Staubli VAL3: ROBERT_TP6.pjx

--- ROBERT_TP6.pjx ---
Parameters version=s7.9 stackSize=5000 millimeterUnit=true
Program file=Poche.pgx
Program file=start.pgx
Program file=stop.pgx
Data file=ROBERT_TP6.dtx

--- ROBERT_TP6.dtx ---
mdesc mRapide100On
mdesc mUsinage20Off = {vel=20, blend=off}
jointRx jStart = {j1=-13.1554864532824, j2=52.8057266959055, j3=128.56179776802, j4=166.840895901009, j5=91.3316286241402, j6=-180.311296989427}
tool tBroche = {x=169.400168374358, y=5.67105066906493E-05, z=47.7499999146672, ry=90, rz=90, fatherId=flange[0], ioLink=valve1}
num nDiametreFraise = 10
frame fPiece = {x=527.606812, y=-37.435701, z=-438.0625, rx=180, rz=-90, fatherId=world[0]}
pointRx pStartUsinage = {x=25, y=25, fatherId=fPiece[0]}
jointRx jChangeOutil = {j1=-4.70104777967739, j2=85.6578357974361, j3=60.0632848818122, j4=174.316678572801, j5=55.8523989241203, j6=-80.7639740285582}
trsf trAppro = {z=-22}
num nPasseRadiale
mdesc mUsinage5Off = {vel=5, blend=off}

--- start.pgx ---
program start()
begin
  resetMotion()
  movej(jStart, tBroche, mRapide100On)

  call Poche(pStartUsinage, nDiametreFraise, 7, 4, 100, 50, 20)

  movej(jChangeOutil, tBroche, mRapide100On)
  waitEndMove()
end

--- Poche.pgx ---
program Poche(pointRx x_pStartPoint, num x_nDiametreTool, num x_nPasseAxiale, num x_nPasseRadiale, num x_nDimX, num x_nDimY, num x_nDimZ)
  local num l_nIndex
  local pointRx l_pPoint[5]
  local num l_nIndex2
  local num l_nN
  local num l_nLongueurCote
  local num l_nIndex3
  local num l_nM
  local num l_nProfondeur
begin
  logMsg("Beginning...")

  l_nProfondeur = x_nDimZ

  l_nN = roundDown((x_nDimX-x_nDiametreTool-x_nPasseRadiale)/(2*x_nPasseRadiale)+1)
  l_nM = roundDown(l_nProfondeur/(x_nPasseAxiale))

  for l_nIndex3 = 1 to l_nM
    logMsg("New passe...")
    if l_nIndex3 == l_nM
      l_pPoint[0] = appro(x_pStartPoint,{x_nDiametreTool/2,x_nDiametreTool/2,l_nProfondeur,0,0,0})
    else
      l_pPoint[0] = appro(x_pStartPoint,{x_nDiametreTool/2,x_nDiametreTool/2,l_nIndex3 * x_nPasseAxiale,0,0,0})
    endIf
    movej(appro(l_pPoint[0],trAppro), tBroche, mRapide100On)

    movel(l_pPoint[0], tBroche, mUsinage20Off)

    //------------------------------------- Forme centrale ------------------------------------------------
    for l_nIndex = 0 to l_nN - 1
      l_pPoint[1] = compose(l_pPoint[0], fPiece, {l_nIndex*2*x_nPasseRadiale,0,0,0,0,0})
      l_pPoint[2] = compose(l_pPoint[1], fPiece, {0,x_nDimY - x_nDiametreTool,0,0,0,0})
      l_pPoint[3] = compose(l_pPoint[2], fPiece, {x_nPasseRadiale,0,0,0,0,0})
      l_pPoint[4] = compose(l_pPoint[3], fPiece, {0,-(x_nDimY - x_nDiametreTool),0,0,0,0})

      for l_nIndex2 = 1 to 4
        movel(l_pPoint[l_nIndex2], tBroche, mUsinage20Off)
      endFor
    endFor
    logMsg("Last 'U'")
    l_pPoint[1] = compose(l_pPoint[0], fPiece, {(x_nDimX - x_nDiametreTool) -  x_nPasseRadiale,0,0,0,0,0})
    l_pPoint[2] = compose(l_pPoint[1], fPiece, {0,x_nDimY - x_nDiametreTool,0,0,0,0})
    l_pPoint[3] = compose(l_pPoint[2], fPiece, {x_nPasseRadiale,0,0,0,0,0})
    l_pPoint[4] = compose(l_pPoint[3], fPiece, {0,-(x_nDimY - x_nDiametreTool),0,0,0,0})

    for l_nIndex2 = 1 to 4
      movel(l_pPoint[l_nIndex2], tBroche, mUsinage20Off)
    endFor

    //------------------------------------- Forme contours ------------------------------------------------

    movel(l_pPoint[0], tBroche, mUsinage20Off)
    movel(appro(l_pPoint[0],trAppro), tBroche, mUsinage20Off)

    l_pPoint[1] = compose(l_pPoint[0], fPiece, {0,x_nDimY - x_nDiametreTool,0,0,0,0})
    l_pPoint[2] = compose(l_pPoint[1], fPiece, {x_nDimX - x_nDiametreTool,0,0,0,0,0})

    movej(appro(l_pPoint[1], trAppro), tBroche, mRapide100On)
    movel(l_pPoint[1], tBroche, mUsinage20Off)
    movel(l_pPoint[2], tBroche, mUsinage20Off)
    movel(appro(l_pPoint[2], trAppro), tBroche, mUsinage20Off)
  endFor
  movej(appro(l_pPoint[0],trAppro), tBroche, mRapide100On)
  logMsg("Program ended.")
end
